TEXTLIST EL1904_M_2
  1 = 'shuttle crash_L' | chinese: '车头防撞L' | Chinese: '车头防撞L'
  2 = 'shuttle crash_R' | chinese: '车头防撞R' | Chinese: '车头防撞R'
  3 = 'interlock_in_cover' | chinese: 'INPUT_透明盖' | Chinese: 'INPUT_透明盖'
  4 = 'interlock_in_cover' | chinese: 'INPUT_透明盖' | Chinese: 'INPUT_透明盖'
   = ''
END_TEXTLIST

(* stored: Version 1.1.0.1, ProductVersion 3.1.4024.11
   TextList EL1904_M_2: Id {dd7a3a63-ab19-439d-b5bf-c41ecbf115c0} *)
